  994 = 'S5_Prompts Default 994' | German: 'S5_Prompts German 994' | French: 'S5_Prompts French 994'
  995 = 'S5_Prompts Default 995' | German: 'S5_Prompts German 995' | French: 'S5_Prompts French 995'
  996 = 'S5_Prompts Default 996' | German: 'S5_Prompts German 996' | French: 'S5_Prompts French 996'
  997 = 'S5_Prompts Default 997' | German: 'S5_Prompts German 997' | French: 'S5_Prompts French 997'
  998 = 'S5_Prompts Default 998' | German: 'S5_Prompts German 998' | French: 'S5_Prompts French 998'
  999 = 'S5_Prompts Default 999' | German: 'S5_Prompts German 999' | French: 'S5_Prompts French 999'
  1000 = 'S5_Prompts Default 1000' | German: 'S5_Prompts German 1000' | French: 'S5_Prompts French 1000'
   = ''
END_TEXTLIST

(* stored: Version 1.1.0.1, ProductVersion 3.1.4024.12
   TextList S5_Prompts: Id {123ee555-c1dd-4a67-9c47-c4b87b3503ba} *)
